TYPE E_STATE_CA :
(
	Docking := 0,
	Undocking,
	Relocation,
	Driving
);
END_TYPE

(* stored: Version 1.1.0.1, ProductVersion 3.1.4024.11
   DUT E_STATE_CA: Id {88babce0-eeae-41d2-a8d4-b8a5d975584a} *)
